Universal Robots URScript: step2c_aggressive_search5_guard20_line1ms_alpha70_vlim5_v1.script

# Step2C aggressive: 5 mm/s t10ms search with 20 N raw normal guard + 0.10s ramp then 1ms signed-Fz closed-loop line run; TP-openable package.
# VERSION: 2026-06-08T1159HKT_STEP2C_AGGRESSIVE_SEARCH5_GUARD20_LINE1MS_ALPHA70_VLIM5_V1
# GENERATED_AT_LOCAL: 2026-06-08T11:59:19+0800
# BEHAVIOR: wait for Kunwei bridge; align to old reference orientation; move to
# old contact-start XY; move to old contact Z + 100 mm; search downward with
# speedl([0,0,-0.005,0,0,0], a=0.500, t=0.010) until raw signed Fz <= -2 N.
# After contact, continue into the 63.58 mm line segment at 10 mm/s. The first 0.10 s of line control uses 10 ms speedl holds, then line control switches to 1 ms holds.
# Aggressive normal Z correction targets signed Fz ~= -target_force_abs, where the bridge
# normally writes target_force_abs=5 N into input register 29.
# Raw contact triggers and safety guards remain unfiltered; only controller
# normal-velocity input uses a light force filter. No UR zero_ftsensor, no
# Kunwei tare/config write, no TCP/payload write, and no output register 34.
# Frequency contract: Kunwei raw may be about 1 kHz; RTDE handoff is requested
# at 500 Hz; search speedl motion gate uses 10 ms holds at 5 mm/s; line control switches to 1 ms holds after 0.10 s, but this must be measured before calling it 500 Hz authority.

def codex_abs(x):
  if x < 0.0:
    return -x
  end
  return x
end

def codex_clamp(x, lo, hi):
  if x < lo:
    return lo
  elif x > hi:
    return hi
  end
  return x
end

def codex_wait_for_sensor_ok(timeout_s):
  local dt = 0.002
  local t = 0.0
  while t < timeout_s:
    if read_input_float_register(27) > 0.5:
      return True
    end
    sync()
    t = t + dt
  end
  return False
end

def codex_wait_for_fresh_heartbeat(timeout_s):
  local dt = 0.002
  local t = 0.0
  local initial_heartbeat = read_input_float_register(26)
  local current_heartbeat = initial_heartbeat
  while t < timeout_s:
    current_heartbeat = read_input_float_register(26)
    write_output_float_register(26, current_heartbeat)
    write_output_float_register(35, 20.5)
    if read_input_float_register(27) > 0.5 and current_heartbeat != initial_heartbeat:
      return True
    end
    sync()
    t = t + dt
  end
  return False
end

def codex_step2_guard_stop_reason():
  local normal_force = read_input_float_register(24)
  local force_norm = read_input_float_register(25)
  local sensor_ok = read_input_float_register(27)
  local stop_request = read_input_float_register(28)
  local torque_norm = read_input_float_register(30)
  if sensor_ok < 0.5:
    return 3.0
  elif stop_request > 0.5:
    return 4.0
  elif codex_abs(normal_force) > 20.0:
    return 5.0
  elif force_norm > 50.0:
    return 6.0
  elif torque_norm > 0.6:
    return 7.0
  end
  return 0.0
end

def codex_write_echo(stop_reason, progress_m, correction_m, commanded_z_m_s):
  write_output_float_register(24, read_input_float_register(24))
  write_output_float_register(25, read_input_float_register(25))
  write_output_float_register(26, read_input_float_register(26))
  write_output_float_register(27, read_input_float_register(27))
  write_output_float_register(28, read_input_float_register(28))
  write_output_float_register(29, read_input_float_register(29))
  write_output_float_register(30, stop_reason)
  write_output_float_register(31, progress_m)
  write_output_float_register(32, correction_m)
  write_output_float_register(33, commanded_z_m_s)
end

def codex_step2c_full():
  local ux = 0.679764156
  local uy = -0.733430768
  local entry_x = 0.446585764
  local entry_y = 0.226717001
  local old_contact_z = 0.020279919
  local entry_z = old_contact_z + 0.100
  local ref_rx = 3.141572714
  local ref_ry = -0.000026465
  local ref_rz = -0.000024158
  local approach_speed_m_s = 0.080
  local approach_z_speed_m_s = 0.080
  local search_speed_m_s = -0.005
  local search_accel_m_s2 = 0.500
  local search_hold_s = 0.010
  local trigger_normal_force_n = -2.0
  local max_search_down_m = 0.110
  local stale_limit_s = 0.100
  local search_runtime_limit_s = 65.0
  local tangent_speed_m_s = 0.010
  local path_length_m = 0.06358
  local line_accel_m_s2 = 0.500
  local line_hold_s = 0.010
  local line_hold_fast_s = 0.001
  local line_fast_after_s = 0.100
  local line_runtime_limit_s = 15.0
  local target_force_abs_default_n = 5.0
  local normal_velocity_p_gain = 0.0006
  local normal_velocity_i_gain = 0.00008
  local normal_velocity_limit_m_s = 0.005
  local normal_filter_alpha = 0.70
  local integral_error_limit_n_s = 10.0
  local unload_speed_m_s = 0.001
  local unload_force_norm_n = 0.8
  local unload_runtime_limit_s = 10.0
  local retract_z_m = 0.050
  local stop_reason = 0.0
  local contact_triggered = 0
  local max_observed_stale_s = 0.0

  textmsg("codex step2c version 2026-06-08T1159HKT_STEP2C_AGGRESSIVE_SEARCH5_GUARD20_LINE1MS_ALPHA70_VLIM5_V1 start search5_guard20_alpha70_kp0006_vlim5_line1ms_after100ms")
  write_output_float_register(35, 20.0)
  codex_write_echo(0.0, 0.0, 0.0, 0.0)

  if not codex_wait_for_fresh_heartbeat(30.0):
    stop_reason = 3.0
  end

  if stop_reason == 0.0:
    write_output_float_register(35, 21.0)
    local p0 = get_actual_tcp_pose()
    local reference_orientation_pose = p[p0[0], p0[1], p0[2], ref_rx, ref_ry, ref_rz]
    movel(reference_orientation_pose, a=0.030, v=approach_speed_m_s, r=0.0)
    stopl(0.5)
    write_output_float_register(35, 22.0)
    local p1 = get_actual_tcp_pose()
    local entry_xy_pose = p[entry_x, entry_y, p1[2], ref_rx, ref_ry, ref_rz]
    movel(entry_xy_pose, a=0.030, v=approach_speed_m_s, r=0.0)
    stopl(0.5)
    write_output_float_register(35, 23.0)
    local entry_pose = p[entry_x, entry_y, entry_z, ref_rx, ref_ry, ref_rz]
    movel(entry_pose, a=0.030, v=approach_z_speed_m_s, r=0.0)
    stopl(0.5)
    sleep(0.20)
    stop_reason = codex_step2_guard_stop_reason()
  end

  if stop_reason == 0.0:
    write_output_float_register(35, 24.0)
    local search_start = get_actual_tcp_pose()
    local last_heartbeat = read_input_float_register(26)
    local stale_s = 0.0
    local t = 0.0
    while stop_reason == 0.0:
      local heartbeat = read_input_float_register(26)
      local normal_force = read_input_float_register(24)
      local pose_now = get_actual_tcp_pose()
      local search_depth_m = search_start[2] - pose_now[2]

      if heartbeat == last_heartbeat:
        stale_s = stale_s + search_hold_s
        if stale_s > max_observed_stale_s:
          max_observed_stale_s = stale_s
        end
      else:
        stale_s = 0.0
        last_heartbeat = heartbeat
      end

      codex_write_echo(stop_reason, max_observed_stale_s, search_depth_m, search_speed_m_s)

      if stale_s > stale_limit_s:
        stop_reason = 2.0
      else:
        stop_reason = codex_step2_guard_stop_reason()
      end

      if stop_reason == 0.0:
        if normal_force <= trigger_normal_force_n:
          contact_triggered = 1
          stop_reason = 11.0
        elif search_depth_m >= max_search_down_m:
          stop_reason = 8.0
        elif t >= search_runtime_limit_s:
          stop_reason = 10.0
        else:
          speedl([0.0, 0.0, search_speed_m_s, 0.0, 0.0, 0.0], search_accel_m_s2, search_hold_s)
          t = t + search_hold_s
        end
      end
    end
    stopl(0.5)

    if stop_reason == 8.0:
      write_output_float_register(35, 28.0)
      local p_end = get_actual_tcp_pose()
      local retract_pose = p[p_end[0], p_end[1], entry_z, p_end[3], p_end[4], p_end[5]]
      movel(retract_pose, a=0.030, v=0.005, r=0.0)
      stopl(0.5)
    end
  end

  if contact_triggered == 1:
    stop_reason = 0.0
  end

  if stop_reason == 0.0:
    write_output_float_register(35, 25.0)
    local line_start = get_actual_tcp_pose()
    local last_heartbeat2 = read_input_float_register(26)
    local stale_s2 = 0.0
    local t2 = 0.0
    local filtered_normal_force = read_input_float_register(24)
    local integral_error = 0.0
    while stop_reason == 0.0:
      if t2 >= line_fast_after_s:
        line_hold_s = line_hold_fast_s
      end
      local raw_normal_force = read_input_float_register(24)
      local heartbeat2 = read_input_float_register(26)
      local target_force_abs = read_input_float_register(29)
      local pose_line = get_actual_tcp_pose()
      local dx = pose_line[0] - line_start[0]
      local dy = pose_line[1] - line_start[1]
      local progress_m = dx * ux + dy * uy
      local correction_m = pose_line[2] - line_start[2]

      if target_force_abs < 0.1:
        target_force_abs = target_force_abs_default_n
      end

      filtered_normal_force = normal_filter_alpha * raw_normal_force + (1.0 - normal_filter_alpha) * filtered_normal_force
      local force_error = target_force_abs + filtered_normal_force
      integral_error = codex_clamp(integral_error + force_error * line_hold_s, -integral_error_limit_n_s, integral_error_limit_n_s)
      local normal_velocity = 0.0 - codex_clamp(normal_velocity_p_gain * force_error + normal_velocity_i_gain * integral_error, -normal_velocity_limit_m_s, normal_velocity_limit_m_s)

      if heartbeat2 == last_heartbeat2:
        stale_s2 = stale_s2 + line_hold_s
      else:
        stale_s2 = 0.0
        last_heartbeat2 = heartbeat2
      end

      codex_write_echo(stop_reason, progress_m, correction_m, normal_velocity)

      if stale_s2 > stale_limit_s:
        stop_reason = 2.0
      else:
        stop_reason = codex_step2_guard_stop_reason()
      end

      if stop_reason == 0.0:
        if codex_abs(correction_m) > 0.008:
          stop_reason = 8.0
        elif progress_m < -0.003 or progress_m > 0.067:
          stop_reason = 9.0
        elif t2 >= line_runtime_limit_s:
          stop_reason = 10.0
        elif progress_m >= path_length_m:
          stop_reason = 1.0
        else:
          speedl([ux * tangent_speed_m_s, uy * tangent_speed_m_s, normal_velocity, 0.0, 0.0, 0.0], line_accel_m_s2, line_hold_s)
          t2 = t2 + line_hold_s
        end
      end
    end
    stopl(0.5)
  end

  if stop_reason == 1.0:
    write_output_float_register(35, 26.0)
    local unload_start = get_actual_tcp_pose()
    local t3 = 0.0
    while t3 < unload_runtime_limit_s and read_input_float_register(25) > unload_force_norm_n:
      local unload_pose = get_actual_tcp_pose()
      local unload_m = unload_pose[2] - unload_start[2]
      codex_write_echo(stop_reason, path_length_m, unload_m, unload_speed_m_s)
      if unload_m > 0.008:
        t3 = unload_runtime_limit_s
      else:
        speedl([0.0, 0.0, unload_speed_m_s, 0.0, 0.0, 0.0], line_accel_m_s2, line_hold_s)
        t3 = t3 + line_hold_s
      end
    end
    stopl(0.5)
    write_output_float_register(35, 27.0)
    local retract_start = get_actual_tcp_pose()
    local retract_pose2 = p[retract_start[0], retract_start[1], retract_start[2] + retract_z_m, retract_start[3], retract_start[4], retract_start[5]]
    movel(retract_pose2, a=0.030, v=0.005, r=0.0)
    stopl(0.5)
  end

  write_output_float_register(30, stop_reason)
  write_output_float_register(31, max_observed_stale_s)
  write_output_float_register(35, 29.0)
  textmsg("codex step2c version 2026-06-08T1159HKT_STEP2C_AGGRESSIVE_SEARCH5_GUARD20_LINE1MS_ALPHA70_VLIM5_V1 stop reason:", stop_reason)
end

codex_step2c_full()
